PROGRAM SignalHandler
VAR
END_VAR

END_PROGRAM

(* stored: Version 1.1.0.1, ProductVersion 3.1.4022.16
   POU SignalHandler: Id {8d1c351c-c5f8-4138-91c0-bf23a590a776}, SpecialFunc None *)
